{attribute 'qualified_only'}
VAR_GLOBAL
END_VAR

(* stored: Version 1.1.0.1, ProductVersion 3.1.4022.7
   GVL GVL_06_Output_Servo_Motor_Shelf_Z: Id {3a09d9b5-2f85-4b90-bbb6-7a591a0924b3} *)
